SUBAPPLICATION Uebung_006e2_AX (* RS-Flip-Flop mit 2x IXA *)
  (* Standard: 61499-2; Description: Copyright (c) 2023 Meisterschulen am Ostbahnhof This program and the accompanying materials are made available under the terms of the Eclipse Public License 2.0 which is available at https://www.eclipse.org/legal/epl-2.0/ SPDX-License-Identifier: EPL-2.0 *)
  (* Version 1.0, 2023-10-23, Franz Höpfinger, Meisterschulen am Ostbahnhof, initial API and implementation and/or initial documentation *)
  PACKAGE Uebungen;
  IMPORT logiBUS::io::DI::logiBUS_DI::Input_I1;
  IMPORT logiBUS::io::DI::logiBUS_DI::Input_I2;
  IMPORT logiBUS::io::DQ::logiBUS_DO::Output_Q1;
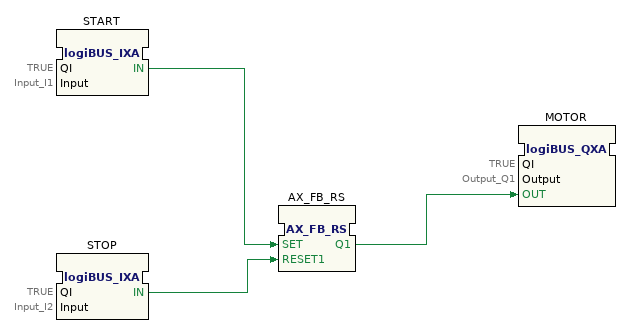
  FBS
    MOTOR : logiBUS::io::DQ::logiBUS_QXA(QI := TRUE, Output := Output_Q1);
    START : logiBUS::io::DI::logiBUS_IXA(QI := TRUE, Input := Input_I1);
    STOP : logiBUS::io::DI::logiBUS_IXA(QI := TRUE, Input := Input_I2);
    AX_FB_RS : adapter::iec61131::bistableElements::AX_FB_RS;
  END_FBS
  ADAPTER_CONNECTIONS
    AX_FB_RS.Q1 TO MOTOR.OUT;
    START.IN TO AX_FB_RS.SET;
    STOP.IN TO AX_FB_RS.RESET1;
  END_CONNECTIONS
END_SUBAPPLICATION
